Staubli VAL3: addActionTime.pgx

public program addActionTime(ActionItem& x_aAction[] (dimensions=1))
  local num l_nSize[2]
begin
  // mutex
  setMutex(bLogMutex)
  // add one action with the timing
  if x_aAction.iInstr.sType==""
    // init
    aActionTime=x_aAction
  else
    // insert
    append(aActionTime)
    aActionTime[size(aActionTime)-1]=x_aAction
    aActionTime[size(aActionTime)-1].nTimeId=clock()-nClockAction
  endIf
  // update
  nClockAction=clock()
  //
  bLogMutex=false
end
